{attribute 'qualified_only'}
{attribute 'strict'}
TYPE ENUM_SeqSM :
(
	Once		:=0, //(Lights, Dry Contacts)
	OnceDC		:=1, // Dry Contact (HVAC)
	Twice		:=2 //(Motors)
);
END_TYPE

(* stored: Version 1.1.0.1, ProductVersion 3.1.4024.9
   DUT ENUM_SeqSM: Id {f017f8af-f1d7-4e02-a4f5-e19b8d3a4417} *)
